// TIA Portal V19 export
DATA_BLOCK "Projekt2B_RobotGrinder_DB"   // DB1
// stored: InstanceOfName Projekt2B_RobotGrinder, InstanceOfType FB
"Projekt2B_RobotGrinder"
   // VAR_INPUT
   //    Emergency_Stop_Status_150K1 : Bool;
   //    Sensor_102B2 : Bool;
   //    Sensor_102B3 : Bool;
   //    Sensor_102B4 : Bool;
   //    Sensor_102B5 : Bool;
   //    Sensor_102B6 : Bool;
   //    Reset : Bool;
   // END_VAR
   // VAR_OUTPUT
   //    Valve_106Q6 : Bool;
   //    Motor_4Q3 : Bool;
   //    Motor_4Q5 : Bool;
   //    Motor_6Q1 : Bool;
   //    Motor_6Q3 : Bool;
   //    Reset_Safety_150K1 : Bool;
   // END_VAR
BEGIN
END_DATA_BLOCK
